ABB RobotStudio station: xhruby26_pick_n_place.rspag

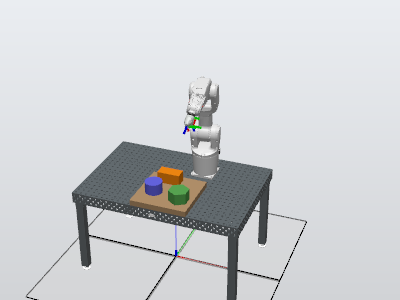
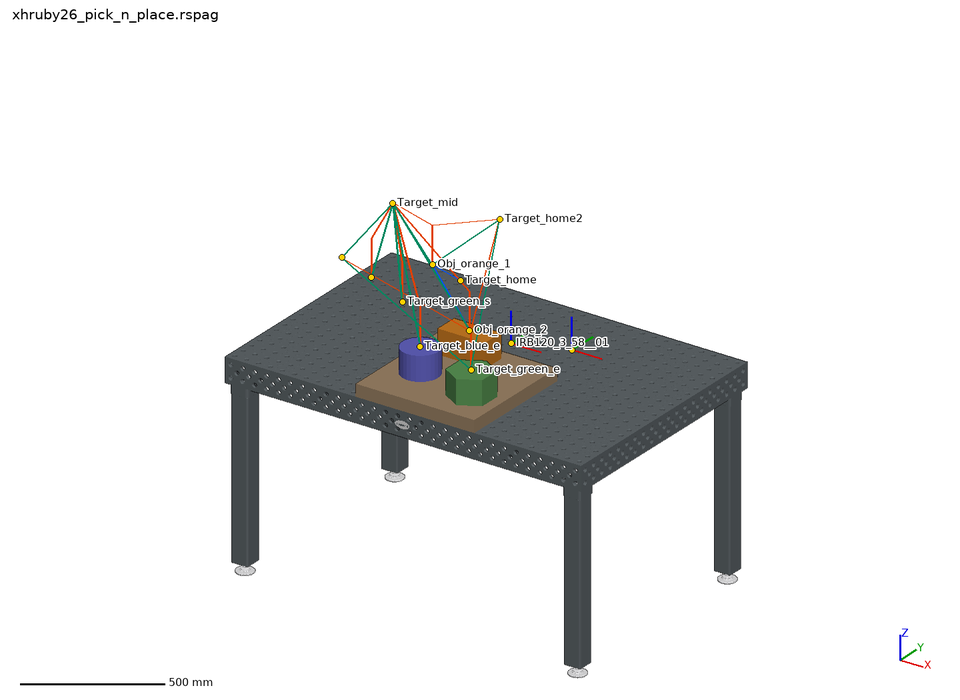
[picture v1: parts stored in the station drawn from their meshes, with robot base, taught points and paths (robot models come from the ABB library and are not in the file)]
--- station ---
Station Solution_1_Tutorial (saved by RobotStudio 22.3.10190.2)
Controller Controller2, task T_ROB1: task frame (RAPID world) sits at (200, 230, 830) mm, rotated rx 0 ry 0 rz -90 deg in the station
Controller Controller1, task T_ROB1: task frame (RAPID world) sits at (0, 150, 830) mm, rotated rx 0 ry 0 rz -90 deg in the station
Controller Controller1
  mechanical unit ROB_1: IRB120_3_58__01, 6 joints, base frame (0, 0, 0) mm
Controller Controller2
  mechanical unit ROB_1: IRB1200_5_90_STD_03_2, 6 joints, base frame (0, 0, 0) mm
Layout (positions relative to the parent item):
  - table [part] at (-200, -500, 830) mm, size 500 x 500 x 50 mm
  - object_1 [part] at (-200, -500, 830) mm, size 200 x 100 x 150 mm
  - object_2 [part] at (-200, -500, 830) mm, size 149.5 x 149.7 x 150 mm
  - object_3 [part] at (-200, -500, 830) mm, size 155.5 x 179.5 x 150 mm
  - siegmund_1500_1000 [part], size 1500 x 1010.3 x 830 mm
  - object_11 [part] at (-200, -500, 830) mm, size 200 x 100 x 150 mm
  - object_22 [part] at (-200, -500, 830) mm, size 149.5 x 149.7 x 150 mm
  - object_33 [part] at (-200, -500, 830) mm, size 155.5 x 179.5 x 150 mm
  - IRB120_3_58__01 [mechanism, from Robots\IRB120_3_58_G_01.rslib] at (0, 150, 830) mm, rotated rx 0 ry 0 rz -90 deg; joint values [0, 0, 0, 0, 1.5708, 0] (rad or m)
  - smc_gripper [mechanism, from Libraries\smc_gripper.rslib] at (0, -152, 1388) mm, rotated rx 180 ry 0 rz 90 deg
  - Positioner [smart component, from Components\Positioner.rslib] at (-600, -150, 830) mm
      properties: Object=object_1; Position=[-0.6 -0.15 0.83]; Orientation=[0 0 0]; Reference=Global; ReferenceObject=(none)
  - Attacher [smart component, from Components\Attacher.rslib]
      properties: Parent=smc_gripper; Flange=0; Child=object_1; Mount=false; Offset=[0 0 0]; Orientation=[0 0 0]
  - Detacher [smart component, from Components\Detacher.rslib]
      properties: Child=object_1; KeepPosition=true
  - IRB1200_5_90_STD_03_2 [mechanism, from %ABB.RobotStudio.Models.IRB1200%\IRB1200_5_90_STD_03.rslib] at (200, 230, 830) mm, rotated rx 0 ry 0 rz -90 deg; joint values [0.1861, 0.2029, -0.2233, -0.3005, 0.5722, 0.3487] (rad or m)
  - Smart_Gripper_Servo_One_Vacuum_2 [mechanism, from Tools\ABB_Smart_Gripper_Servo_One_Vacuum.rslib] at (300, -372.01, 1678.1) mm, rotated rx -180 ry 60 rz 90 deg; joint values [0] (rad or m)
  - Attacher_2 [smart component, from Components\Attacher.rslib]
      properties: Parent=Smart_Gripper_Servo_One_Vacuum_2; Flange=0; Child=object_1; Mount=false; Offset=[0 0 0]; Orientation=[0 0 0]
  - Attacher_3 [smart component, from Components\Attacher.rslib]
      properties: Parent=Smart_Gripper_Servo_One_Vacuum_2; Flange=0; Child=object_2; Mount=false; Offset=[0 0 0]; Orientation=[0 0 0]
  - Attacher_4 [smart component, from Components\Attacher.rslib]
      properties: Parent=Smart_Gripper_Servo_One_Vacuum_2; Flange=0; Child=object_3; Mount=false; Offset=[0 0 0]; Orientation=[0 0 0]
  - Detacher_2 [smart component, from Components\Detacher.rslib]
      properties: Child=object_1; KeepPosition=true
  - Detacher_3 [smart component, from Components\Detacher.rslib]
      properties: Child=object_2; KeepPosition=true
  - Detacher_4 [smart component, from Components\Detacher.rslib]
      properties: Child=object_3; KeepPosition=true
  - Positioner_2 [smart component, from Components\Positioner.rslib]
      properties: Object=object_1; Position=[-0.6 -0.15 0.83]; Orientation=[0 0 0]; Reference=Global; ReferenceObject=(none)
  - Positioner_3 [smart component, from Components\Positioner.rslib]
      properties: Object=object_3; Position=[-0.7 -0.2 0.83]; Orientation=[0 0 0]; Reference=Global; ReferenceObject=(none)
  - Positioner_4 [smart component, from Components\Positioner.rslib]
      properties: Object=object_2; Position=[-0.65 -0.15 0.83]; Orientation=[0 0 0]; Reference=Global; ReferenceObject=(none)
Attachment: smc_gripper is attached to IRB120_3_58__01 / Link6
Attachment: Smart_Gripper_Servo_One_Vacuum_2 is attached to IRB1200_5_90_STD_03_2 / Link6
Collision set CollisionSet_1: object_1 against object_2, object_3, near miss 0 m
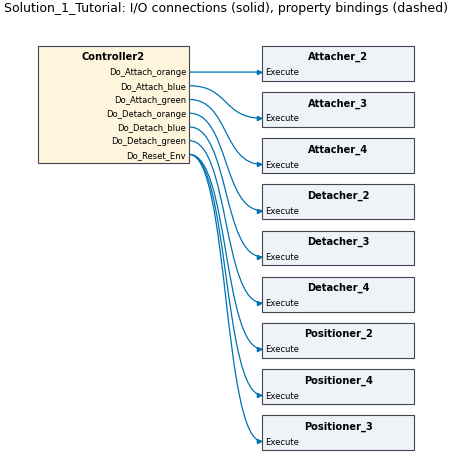
Station logic (signal -> signal, property => property):
  Controller2.Do_Attach_orange -> Attacher_2.Execute
  Controller2.Do_Attach_blue -> Attacher_3.Execute
  Controller2.Do_Attach_green -> Attacher_4.Execute
  Controller2.Do_Detach_orange -> Detacher_2.Execute
  Controller2.Do_Detach_blue -> Detacher_3.Execute
  Controller2.Do_Detach_green -> Detacher_4.Execute
  Controller2.Do_Reset_Env -> Positioner_2.Execute
  Controller2.Do_Reset_Env -> Positioner_4.Execute
  Controller2.Do_Reset_Env -> Positioner_3.Execute

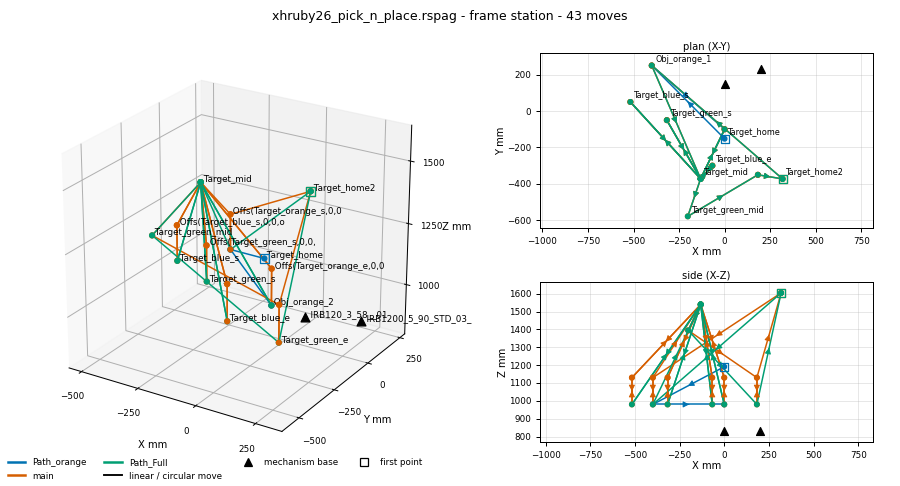
[picture p0: tool path of xhruby26_pick_n_place.rspag in frame station, 43 of 43 moves have a stored position in this frame; points joined in program order, loops and branches not executed]
--- Backups/Controller1/RAPID/TASK1/PROGMOD/CalibData.mod ---
MODULE CalibData
    PERS tooldata smc_gripper:=[TRUE,[[0,0.004,197.001],[1,0,0,0]],[1,[0.207,-0.496,71.18],[1,0,0,0],0,0,0]];
ENDMODULE

--- Backups/Controller1/RAPID/TASK1/PROGMOD/Module1.mod ---
MODULE Module1
    CONST robtarget Target_home:=[[302,0.004004008,360.999],[0,-0.000000007,1,0],[0,0,-1,0],[9E+09,9E+09,9E+09,9E+09,9E+09,9E+09]];
    CONST robtarget Obj_orange_1:=[[-100,-400,150],[0,-0.000000007,1,0],[-2,0,-2,0],[9E+09,9E+09,9E+09,9E+09,9E+09,9E+09]];
    CONST robtarget Obj_orange_2:=[[250,0,150],[0,-0.000000007,1,0],[-1,0,-1,0],[9E+09,9E+09,9E+09,9E+09,9E+09,9E+09]];

    VAR num offset_z := 200;

    PROC main()
        ! Reset ENV


        !PulseDO  Do_Detach_Obj1;

        !PulseDO Do_Reset_Obj1; !Na dobu jednoho cyklu se dostane 1


        ! Home position
        !MoveJ Target_home,v100,z100,smc_gripper\WObj:=wobj0;

        ! Pick object
        !MoveL offs(Obj_orange_1,0,0,100),v100,fine,smc_gripper\WObj:=wobj0;
        !MoveL offs(Obj_orange_1,0,0,0),v100,fine,smc_gripper\WObj:=wobj0;
        !..
        !PulseDO Do_Attach_Obj1;
        !WaitTime 1.0;

        !MoveL offs(Obj_orange_1,0,0,100),v100,fine,smc_gripper\WObj:=wobj0;

        ! Home position
        !MoveJ Target_home,v100,z100,smc_gripper\WObj:=wobj0;

        ! Place object
        !MoveL offs(Obj_orange_2,0,0,100),v100,fine,smc_gripper\WObj:=wobj0;
        !MoveL offs(Obj_orange_2,0,0,0),v100,fine,smc_gripper\WObj:=wobj0;
        !...
        !PulseDO Do_Detach_Obj1;
        !WaitTime 1.0;

        !MoveL offs(Obj_orange_2,0,0,100),v100,fine,smc_gripper\WObj:=wobj0;

        ! Home position
        !MoveJ Target_home,v100,z100,smc_gripper\WObj:=wobj0;


    ENDPROC

    PROC Path_orange()
        MoveL Target_home,v100,z100,smc_gripper\WObj:=wobj0;
        MoveL Obj_orange_1,v100,z100,smc_gripper\WObj:=wobj0;
        MoveL Obj_orange_2,v100,z100,smc_gripper\WObj:=wobj0;
    ENDPROC
ENDMODULE

--- Backups/Controller2/RAPID/TASK1/PROGMOD/CalibData.mod ---
MODULE CalibData
    PERS tooldata Servo:=[TRUE,[[0,0,84],[1,0,0,0]],[0.226,[8.9,12.3,48.7],[1,0,0,0],0.00021,0.00024,0.00009]];
    PERS tooldata VaccumOne:=[TRUE,[[63.5,18.5,37.5],[0.707106781,0,0.707106781,0]],[0.226,[8.9,12.3,48.7],[1,0,0,0],0.00021,0.00024,0.00009]];
ENDMODULE

--- Backups/Controller2/RAPID/TASK1/PROGMOD/Module1.mod ---
MODULE Module1

    !CONST robtarget Target_home2[];

    VAR num offset_z := 150;

    CONST robtarget Target_home2:=[[602.740035752,118.5,774.35738686],[0.258819045,0,-0.965925826,0],[0,-1,0,0],[9E+09,9E+09,9E+09,9E+09,9E+09,9E+09]];
    CONST robtarget Target_orange_s:=[[-20,-600,150],[0,0.707106781,0.707106781,0],[-2,-3,2,0],[9E+09,9E+09,9E+09,9E+09,9E+09,9E+09]];
    CONST robtarget Target_mid:=[[601.951809945,-331.6854758,709.532778121],[0.021497552,0.351404997,0.935941898,-0.008071385],[-1,-2,1,0],[9E+09,9E+09,9E+09,9E+09,9E+09,9E+09]];
    CONST robtarget Target_orange_e:=[[330,-200,150],[0,0.707106781,0.707106781,0],[-1,-2,2,0],[9E+09,9E+09,9E+09,9E+09,9E+09,9E+09]];
    CONST robtarget Target_blue_s:=[[180,-717.298,150],[0,0.707106781,0.707106781,0],[-1,-2,1,0],[9E+09,9E+09,9E+09,9E+09,9E+09,9E+09]];
    CONST robtarget Target_blue_e:=[[530,-267.298,150],[0,0.707106781,0.707106781,0],[-1,-2,1,0],[9E+09,9E+09,9E+09,9E+09,9E+09,9E+09]];
    CONST robtarget Target_green_s:=[[280,-517.298,150],[0,0.707106781,0.707106781,0],[-1,-2,1,0],[9E+09,9E+09,9E+09,9E+09,9E+09,9E+09]];
    CONST robtarget Target_green_e:=[[580,-17.298,150],[0,0.707106781,0.707106781,0],[0,-1,1,0],[9E+09,9E+09,9E+09,9E+09,9E+09,9E+09]];
    CONST robtarget Target_green_mid:=[[808.25237185,-402.222286895,564.619533658],[0.027532045,0.307140578,0.951224276,-0.008889816],[-1,-2,1,0],[9E+09,9E+09,9E+09,9E+09,9E+09,9E+09]];

    PROC main()
        ! Reset Environment
        PulseDO Do_Detach_orange;
        PulseDO Do_Detach_blue;
        PulseDO Do_Detach_green;

        PulseDO Do_Reset_Env;

        ! Home Position

        MoveL Target_home2,v150,fine,VaccumOne\WObj:=wobj0;

        ! Pick Orange
        MoveL Offs(Target_orange_s, 0, 0, offset_z),v300,z100,VaccumOne\WObj:=wobj0;
        MoveL Offs(Target_orange_s, 0, 0, 0),v100,fine,VaccumOne\WObj:=wobj0;
        WaitTime 0.5;
        PulseDO Do_Attach_orange;
        WaitTime 0.3;
        MoveL Offs(Target_orange_s, 0, 0, offset_z),v300,z100,VaccumOne\WObj:=wobj0;

        ! Mid Position
        MoveL Target_mid,v300,z200,VaccumOne\WObj:=wobj0;

        ! Place Orange
        MoveL Offs(Target_orange_e, 0, 0, offset_z),v300,z100,VaccumOne\WObj:=wobj0;
        MoveL Offs(Target_orange_e, 0, 0, 0),v50,fine,VaccumOne\WObj:=wobj0;
        WaitTime 0.5;
        PulseDO Do_Detach_orange;
        WaitTime 0.3;
        MoveL Offs(Target_orange_e, 0, 0, offset_z),v300,z100,VaccumOne\WObj:=wobj0;

        ! Mid Position
        MoveL Target_mid,v300,z200,VaccumOne\WObj:=wobj0;

        ! Pick Blue
        MoveL Offs(Target_blue_s, 0, 0, offset_z),v300,z100,VaccumOne\WObj:=wobj0;
        MoveL Offs(Target_blue_s, 0, 0, 0),v100,fine,VaccumOne\WObj:=wobj0;
        WaitTime 0.5;
        PulseDO Do_Attach_blue;
        WaitTime 0.3;
        MoveL Offs(Target_blue_s, 0, 0, offset_z),v300,z100,VaccumOne\WObj:=wobj0;

        ! Mid Position
        MoveL Target_mid,v300,z200,VaccumOne\WObj:=wobj0;

        ! Place Blue
        MoveL Offs(Target_blue_e, 0, 0, offset_z),v300,z100,VaccumOne\WObj:=wobj0;
        MoveL Offs(Target_blue_e, 0, 0, 0),v50,fine,VaccumOne\WObj:=wobj0;
        WaitTime 0.5;
        PulseDO Do_Detach_blue;
        WaitTime 0.3;
        MoveL Offs(Target_blue_e, 0, 0, offset_z),v300,z100,VaccumOne\WObj:=wobj0;

        ! Mid Position
        MoveL Target_mid,v300,z200,VaccumOne\WObj:=wobj0;

        ! Pick Green
        MoveL Offs(Target_green_s, 0, 0, offset_z),v300,z100,VaccumOne\WObj:=wobj0;
        MoveL Offs(Target_green_s, 0, 0, 0),v100,fine,VaccumOne\WObj:=wobj0;
        WaitTime 0.5;
        PulseDO Do_Attach_green;
        WaitTime 0.3;
        MoveL Offs(Target_green_s, 0, 0, offset_z),v300,z100,VaccumOne\WObj:=wobj0;

        ! Mid Position
        MoveL Target_mid,v300,z200,VaccumOne\WObj:=wobj0;
        MoveL Target_green_mid,v300,z200,VaccumOne\WObj:=wobj0;

        ! Place Green
        MoveL Offs(Target_green_e, 0, 0, offset_z),v300,z100,VaccumOne\WObj:=wobj0;
        MoveL Offs(Target_green_e, 0, 0, 0),v50,fine,VaccumOne\WObj:=wobj0;
        WaitTime 0.5;
        PulseDO Do_Detach_green;
        WaitTime 0.3;
        MoveL Offs(Target_green_e, 0, 0, offset_z),v300,z100,VaccumOne\WObj:=wobj0;

        ! Home Position
        MoveL Target_home2,v150,fine,VaccumOne\WObj:=wobj0;


    ENDPROC
    PROC Path_Full()
        MoveL Target_home2,v1000,z100,VaccumOne\WObj:=wobj0;
        MoveL Target_orange_s,v1000,z100,VaccumOne\WObj:=wobj0;
        MoveL Target_mid,v1000,z100,VaccumOne\WObj:=wobj0;
        MoveL Target_orange_e,v1000,z100,VaccumOne\WObj:=wobj0;
        MoveL Target_mid,v1000,z100,VaccumOne\WObj:=wobj0;
        MoveL Target_blue_s,v1000,z100,VaccumOne\WObj:=wobj0;
        MoveL Target_mid,v1000,z100,VaccumOne\WObj:=wobj0;
        MoveL Target_blue_e,v1000,z100,VaccumOne\WObj:=wobj0;
        MoveL Target_mid,v1000,z100,VaccumOne\WObj:=wobj0;
        MoveL Target_green_s,v1000,z100,VaccumOne\WObj:=wobj0;
        MoveL Target_mid,v1000,z100,VaccumOne\WObj:=wobj0;
        MoveL Target_green_mid,v1000,z100,VaccumOne\WObj:=wobj0;
        MoveL Target_green_e,v1000,z100,VaccumOne\WObj:=wobj0;
        MoveL Target_home2,v1000,z100,VaccumOne\WObj:=wobj0;
    ENDPROC
ENDMODULE

--- Backups/Controller1/SYSPAR/EIO.cfg ---
EIO:CFG_1.0:6:1::
#
EIO_SIGNAL:

      -Name "Do_Detach_Obj1" -SignalType "DO"

      -Name "Do_Attach_Obj1" -SignalType "DO"

      -Name "Do_Reset_Obj1" -SignalType "DO"

--- Backups/Controller2/SYSPAR/EIO.cfg ---
EIO:CFG_1.0:6:1::
#
EIO_SIGNAL:

      -Name "Do_Attach_orange" -SignalType "DO"

      -Name "Do_Reset_Env" -SignalType "DO"

      -Name "Do_Detach_orange" -SignalType "DO"

      -Name "Do_Attach_blue" -SignalType "DO"

      -Name "Do_Detach_blue" -SignalType "DO"

      -Name "Do_Attach_green" -SignalType "DO"

      -Name "Do_Detach_green" -SignalType "DO"
